TYPE CmpHMI :
STRUCT
	
	Title : STRING := '';
	Message : STRING := '';
	Timeout : TIME := T#0s;
	InformationOnly :BOOL;
	Trigger : BOOL;
	RespPositive : BOOL;
	RespNegative : BOOL;
	RespTimeout : BOOL;
	HeartbeatOK : BOOL;
	
END_STRUCT
END_TYPE

(* stored: Version 1.1.0.1, ProductVersion 3.1.4024.6
   DUT CmpHMI: Id {2c12cc39-c5ea-4d93-bf0a-704d9da8a5b8} *)
